// TIA Portal V17 export
// export: Created 2023-12-22T15:02:59.0767996Z, ExportSetting WithDefaults, DisplayName Totally Integrated Automation Portal, DisplayVersion V17, DisplayName TIA Portal Openness, DisplayVersion V17, DisplayName TIA Portal Version Control Interface, DisplayVersion V17, DisplayName STEP 7 Professional, DisplayVersion V17, DisplayName STEP 7 Safety, DisplayVersion V17, DisplayName WinCC Advanced, DisplayVersion V17
FUNCTION_BLOCK "Put_Get"   // FB2, LAD
TITLE = ADDR - удаленный PLC
{ S7_Optimized_Access := 'TRUE' }
VERSION : 0.1
// RD - блок в этом PLC
// stored: AutoNumber true, IsIECCheckEnabled false, IsRetainMemResEnabled false, MemoryReserve 100, SetENOAutomatically false, UDAEnableTagReadback false
   VAR
      GET_SKV_1 { S7_SetPoint := 'True'} : GET;
      GET_SKV_2 { S7_SetPoint := 'True'} : GET;
      GET_SKV_3 { S7_SetPoint := 'True'} : GET;
      GET_SKV_12 { S7_SetPoint := 'True'} : GET;
      GET_SKV_13 { S7_SetPoint := 'True'} : GET;
      GET_SKV_14 { S7_SetPoint := 'True'} : GET;
      GET_SKV_15 { S7_SetPoint := 'True'} : GET;
      GET_SKV_20 { S7_SetPoint := 'True'} : GET;
      GET_SKV_21 { S7_SetPoint := 'True'} : GET;
      GET_SKV_22 { S7_SetPoint := 'True'} : GET;
      GET_SKV_23 { S7_SetPoint := 'True'} : GET;
      PUT_SKV_1 { S7_SetPoint := 'True'} : PUT;
      PUT_SKV_2 { S7_SetPoint := 'True'} : PUT;
      PUT_SKV_3 { S7_SetPoint := 'True'} : PUT;
      PUT_SKV_12 { S7_SetPoint := 'True'} : PUT;
      PUT_SKV_13 { S7_SetPoint := 'True'} : PUT;
      PUT_SKV_14 { S7_SetPoint := 'True'} : PUT;
      PUT_SKV_15 { S7_SetPoint := 'True'} : PUT;
      PUT_SKV_20 { S7_SetPoint := 'True'} : PUT;
      PUT_SKV_21 { S7_SetPoint := 'True'} : PUT;
      PUT_SKV_22 { S7_SetPoint := 'True'} : PUT;
      PUT_SKV_23 { S7_SetPoint := 'True'} : PUT;
      GET_SKD2 { S7_SetPoint := 'True'} : GET;
      PUT_SKD2 { S7_SetPoint := 'True'} : PUT;
   END_VAR
   VAR_TEMP   // added for the SCL form of the ladder/FBD networks
      _w1 : Bool;
      _w2 : Bool;
   END_VAR
BEGIN

REGION Network 1: SKV 1
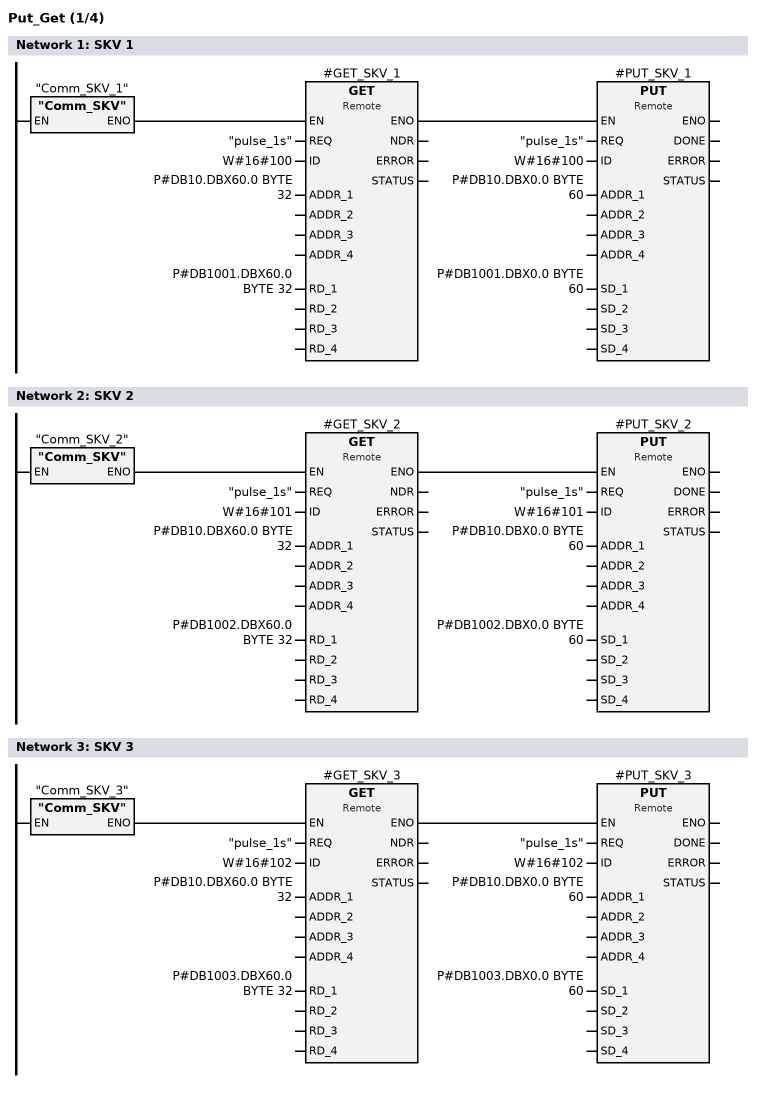
   RUNG wire#powerrail
      "Comm_SKV_1"()
      { S7_Templates := "[remote_type := Remote, local_type := Variant]" } #GET_SKV_1.GET(REQ := "pulse_1s", ID := W#16#100, ADDR_1 := P#DB10.DBX60.0 BYTE 32, ADDR_2 :=, ADDR_3 :=, ADDR_4 :=, RD_1 := P#DB1001.DBX60.0 BYTE 32, RD_2 :=, RD_3 :=, RD_4 :=, NDR =>, ERROR =>, STATUS =>)
      { S7_Templates := "[remote_type := Remote, local_type := Variant]" } #PUT_SKV_1.PUT(REQ := "pulse_1s", ID := W#16#100, ADDR_1 := P#DB10.DBX0.0 BYTE 60, ADDR_2 :=, ADDR_3 :=, ADDR_4 :=, SD_1 := P#DB1001.DBX0.0 BYTE 60, SD_2 :=, SD_3 :=, SD_4 :=, DONE =>, ERROR =>, STATUS =>)
   END_RUNG
   // the same network as SCL:
   "Comm_SKV_1"(ENO => #_w1);   // "Comm_SKV"
   #GET_SKV_1(EN := #_w1,   // GET
              REQ := "pulse_1s",
              ID := W#16#100,
              ADDR_1 := P#DB10.DBX60.0 BYTE 32,
              RD_1 := P#DB1001.DBX60.0 BYTE 32,
              ENO => #_w2);
   IF #_w2 THEN
       #PUT_SKV_1(REQ := "pulse_1s",   // PUT
                  ID := W#16#100,
                  ADDR_1 := P#DB10.DBX0.0 BYTE 60,
                  SD_1 := P#DB1001.DBX0.0 BYTE 60);
   END_IF;
END_REGION

REGION Network 2: SKV 2
   RUNG wire#powerrail
      "Comm_SKV_2"()
      { S7_Templates := "[remote_type := Remote, local_type := Variant]" } #GET_SKV_2.GET(REQ := "pulse_1s", ID := W#16#101, ADDR_1 := P#DB10.DBX60.0 BYTE 32, ADDR_2 :=, ADDR_3 :=, ADDR_4 :=, RD_1 := P#DB1002.DBX60.0 BYTE 32, RD_2 :=, RD_3 :=, RD_4 :=, NDR =>, ERROR =>, STATUS =>)
      { S7_Templates := "[remote_type := Remote, local_type := Variant]" } #PUT_SKV_2.PUT(REQ := "pulse_1s", ID := W#16#101, ADDR_1 := P#DB10.DBX0.0 BYTE 60, ADDR_2 :=, ADDR_3 :=, ADDR_4 :=, SD_1 := P#DB1002.DBX0.0 BYTE 60, SD_2 :=, SD_3 :=, SD_4 :=, DONE =>, ERROR =>, STATUS =>)
   END_RUNG
   // the same network as SCL:
   "Comm_SKV_2"(ENO => #_w1);   // "Comm_SKV"
   #GET_SKV_2(EN := #_w1,   // GET
              REQ := "pulse_1s",
              ID := W#16#101,
              ADDR_1 := P#DB10.DBX60.0 BYTE 32,
              RD_1 := P#DB1002.DBX60.0 BYTE 32,
              ENO => #_w2);
   IF #_w2 THEN
       #PUT_SKV_2(REQ := "pulse_1s",   // PUT
                  ID := W#16#101,
                  ADDR_1 := P#DB10.DBX0.0 BYTE 60,
                  SD_1 := P#DB1002.DBX0.0 BYTE 60);
   END_IF;
END_REGION

REGION Network 3: SKV 3
   RUNG wire#powerrail
      "Comm_SKV_3"()
      { S7_Templates := "[remote_type := Remote, local_type := Variant]" } #GET_SKV_3.GET(REQ := "pulse_1s", ID := W#16#102, ADDR_1 := P#DB10.DBX60.0 BYTE 32, ADDR_2 :=, ADDR_3 :=, ADDR_4 :=, RD_1 := P#DB1003.DBX60.0 BYTE 32, RD_2 :=, RD_3 :=, RD_4 :=, NDR =>, ERROR =>, STATUS =>)
      { S7_Templates := "[remote_type := Remote, local_type := Variant]" } #PUT_SKV_3.PUT(REQ := "pulse_1s", ID := W#16#102, ADDR_1 := P#DB10.DBX0.0 BYTE 60, ADDR_2 :=, ADDR_3 :=, ADDR_4 :=, SD_1 := P#DB1003.DBX0.0 BYTE 60, SD_2 :=, SD_3 :=, SD_4 :=, DONE =>, ERROR =>, STATUS =>)
   END_RUNG
   // the same network as SCL:
   "Comm_SKV_3"(ENO => #_w1);   // "Comm_SKV"
   #GET_SKV_3(EN := #_w1,   // GET
              REQ := "pulse_1s",
              ID := W#16#102,
              ADDR_1 := P#DB10.DBX60.0 BYTE 32,
              RD_1 := P#DB1003.DBX60.0 BYTE 32,
              ENO => #_w2);
   IF #_w2 THEN
       #PUT_SKV_3(REQ := "pulse_1s",   // PUT
                  ID := W#16#102,
                  ADDR_1 := P#DB10.DBX0.0 BYTE 60,
                  SD_1 := P#DB1003.DBX0.0 BYTE 60);
   END_IF;
END_REGION

REGION Network 4: SKV 4
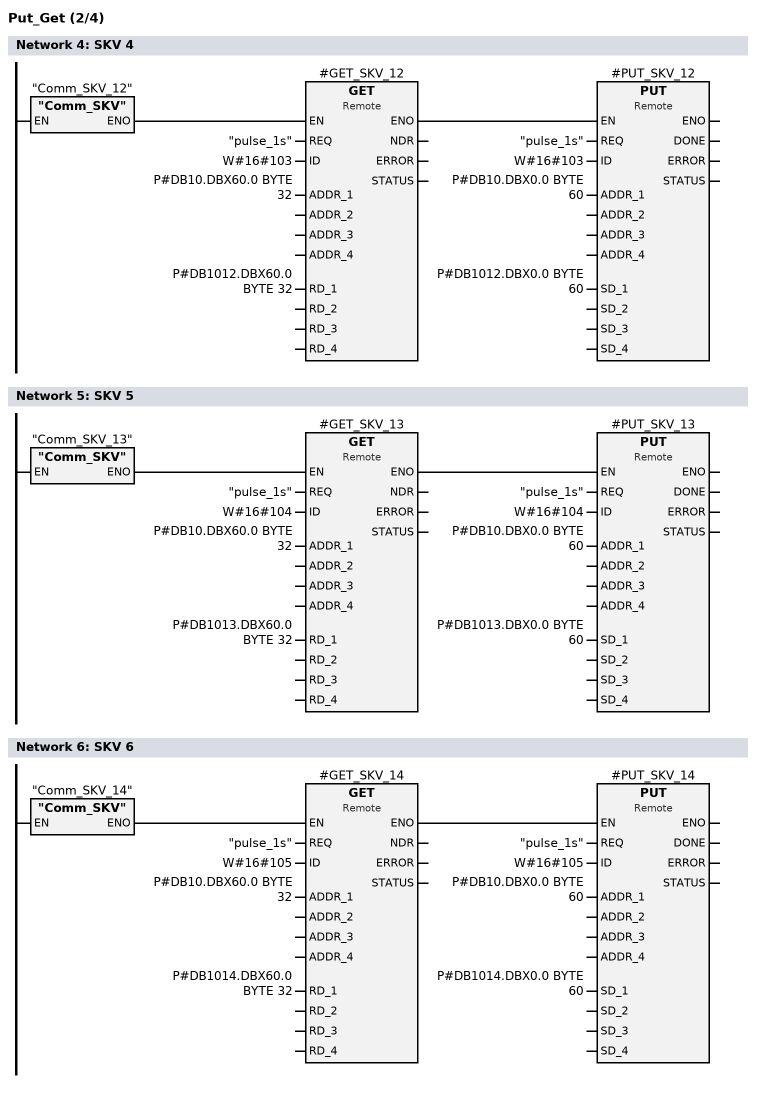
   RUNG wire#powerrail
      "Comm_SKV_12"()
      { S7_Templates := "[remote_type := Remote, local_type := Variant]" } #GET_SKV_12.GET(REQ := "pulse_1s", ID := W#16#103, ADDR_1 := P#DB10.DBX60.0 BYTE 32, ADDR_2 :=, ADDR_3 :=, ADDR_4 :=, RD_1 := P#DB1012.DBX60.0 BYTE 32, RD_2 :=, RD_3 :=, RD_4 :=, NDR =>, ERROR =>, STATUS =>)
      { S7_Templates := "[remote_type := Remote, local_type := Variant]" } #PUT_SKV_12.PUT(REQ := "pulse_1s", ID := W#16#103, ADDR_1 := P#DB10.DBX0.0 BYTE 60, ADDR_2 :=, ADDR_3 :=, ADDR_4 :=, SD_1 := P#DB1012.DBX0.0 BYTE 60, SD_2 :=, SD_3 :=, SD_4 :=, DONE =>, ERROR =>, STATUS =>)
   END_RUNG
   // the same network as SCL:
   "Comm_SKV_12"(ENO => #_w1);   // "Comm_SKV"
   #GET_SKV_12(EN := #_w1,   // GET
               REQ := "pulse_1s",
               ID := W#16#103,
               ADDR_1 := P#DB10.DBX60.0 BYTE 32,
               RD_1 := P#DB1012.DBX60.0 BYTE 32,
               ENO => #_w2);
   IF #_w2 THEN
       #PUT_SKV_12(REQ := "pulse_1s",   // PUT
                   ID := W#16#103,
                   ADDR_1 := P#DB10.DBX0.0 BYTE 60,
                   SD_1 := P#DB1012.DBX0.0 BYTE 60);
   END_IF;
END_REGION

REGION Network 5: SKV 5
   RUNG wire#powerrail
      "Comm_SKV_13"()
      { S7_Templates := "[remote_type := Remote, local_type := Variant]" } #GET_SKV_13.GET(REQ := "pulse_1s", ID := W#16#104, ADDR_1 := P#DB10.DBX60.0 BYTE 32, ADDR_2 :=, ADDR_3 :=, ADDR_4 :=, RD_1 := P#DB1013.DBX60.0 BYTE 32, RD_2 :=, RD_3 :=, RD_4 :=, NDR =>, ERROR =>, STATUS =>)
      { S7_Templates := "[remote_type := Remote, local_type := Variant]" } #PUT_SKV_13.PUT(REQ := "pulse_1s", ID := W#16#104, ADDR_1 := P#DB10.DBX0.0 BYTE 60, ADDR_2 :=, ADDR_3 :=, ADDR_4 :=, SD_1 := P#DB1013.DBX0.0 BYTE 60, SD_2 :=, SD_3 :=, SD_4 :=, DONE =>, ERROR =>, STATUS =>)
   END_RUNG
   // the same network as SCL:
   "Comm_SKV_13"(ENO => #_w1);   // "Comm_SKV"
   #GET_SKV_13(EN := #_w1,   // GET
               REQ := "pulse_1s",
               ID := W#16#104,
               ADDR_1 := P#DB10.DBX60.0 BYTE 32,
               RD_1 := P#DB1013.DBX60.0 BYTE 32,
               ENO => #_w2);
   IF #_w2 THEN
       #PUT_SKV_13(REQ := "pulse_1s",   // PUT
                   ID := W#16#104,
                   ADDR_1 := P#DB10.DBX0.0 BYTE 60,
                   SD_1 := P#DB1013.DBX0.0 BYTE 60);
   END_IF;
END_REGION

REGION Network 6: SKV 6
   RUNG wire#powerrail
      "Comm_SKV_14"()
      { S7_Templates := "[remote_type := Remote, local_type := Variant]" } #GET_SKV_14.GET(REQ := "pulse_1s", ID := W#16#105, ADDR_1 := P#DB10.DBX60.0 BYTE 32, ADDR_2 :=, ADDR_3 :=, ADDR_4 :=, RD_1 := P#DB1014.DBX60.0 BYTE 32, RD_2 :=, RD_3 :=, RD_4 :=, NDR =>, ERROR =>, STATUS =>)
      { S7_Templates := "[remote_type := Remote, local_type := Variant]" } #PUT_SKV_14.PUT(REQ := "pulse_1s", ID := W#16#105, ADDR_1 := P#DB10.DBX0.0 BYTE 60, ADDR_2 :=, ADDR_3 :=, ADDR_4 :=, SD_1 := P#DB1014.DBX0.0 BYTE 60, SD_2 :=, SD_3 :=, SD_4 :=, DONE =>, ERROR =>, STATUS =>)
   END_RUNG
   // the same network as SCL:
   "Comm_SKV_14"(ENO => #_w1);   // "Comm_SKV"
   #GET_SKV_14(EN := #_w1,   // GET
               REQ := "pulse_1s",
               ID := W#16#105,
               ADDR_1 := P#DB10.DBX60.0 BYTE 32,
               RD_1 := P#DB1014.DBX60.0 BYTE 32,
               ENO => #_w2);
   IF #_w2 THEN
       #PUT_SKV_14(REQ := "pulse_1s",   // PUT
                   ID := W#16#105,
                   ADDR_1 := P#DB10.DBX0.0 BYTE 60,
                   SD_1 := P#DB1014.DBX0.0 BYTE 60);
   END_IF;
END_REGION

REGION Network 7: SKV 7
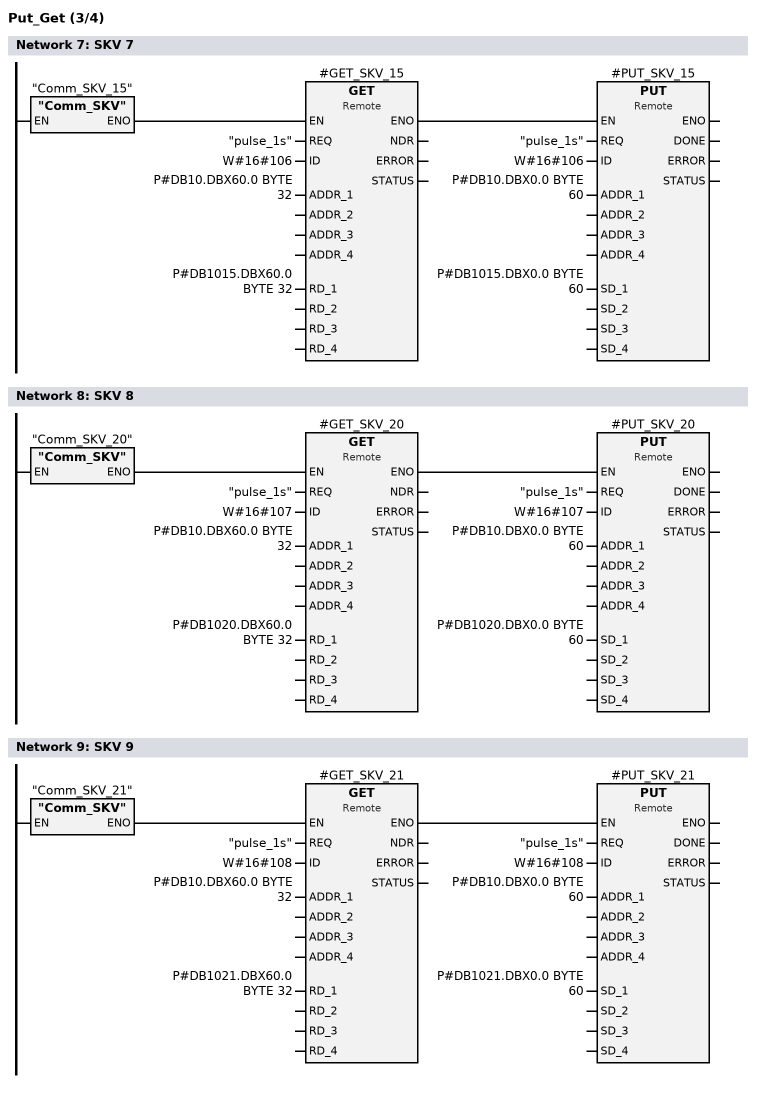
   RUNG wire#powerrail
      "Comm_SKV_15"()
      { S7_Templates := "[remote_type := Remote, local_type := Variant]" } #GET_SKV_15.GET(REQ := "pulse_1s", ID := W#16#106, ADDR_1 := P#DB10.DBX60.0 BYTE 32, ADDR_2 :=, ADDR_3 :=, ADDR_4 :=, RD_1 := P#DB1015.DBX60.0 BYTE 32, RD_2 :=, RD_3 :=, RD_4 :=, NDR =>, ERROR =>, STATUS =>)
      { S7_Templates := "[remote_type := Remote, local_type := Variant]" } #PUT_SKV_15.PUT(REQ := "pulse_1s", ID := W#16#106, ADDR_1 := P#DB10.DBX0.0 BYTE 60, ADDR_2 :=, ADDR_3 :=, ADDR_4 :=, SD_1 := P#DB1015.DBX0.0 BYTE 60, SD_2 :=, SD_3 :=, SD_4 :=, DONE =>, ERROR =>, STATUS =>)
   END_RUNG
   // the same network as SCL:
   "Comm_SKV_15"(ENO => #_w1);   // "Comm_SKV"
   #GET_SKV_15(EN := #_w1,   // GET
               REQ := "pulse_1s",
               ID := W#16#106,
               ADDR_1 := P#DB10.DBX60.0 BYTE 32,
               RD_1 := P#DB1015.DBX60.0 BYTE 32,
               ENO => #_w2);
   IF #_w2 THEN
       #PUT_SKV_15(REQ := "pulse_1s",   // PUT
                   ID := W#16#106,
                   ADDR_1 := P#DB10.DBX0.0 BYTE 60,
                   SD_1 := P#DB1015.DBX0.0 BYTE 60);
   END_IF;
END_REGION

REGION Network 8: SKV 8
   RUNG wire#powerrail
      "Comm_SKV_20"()
      { S7_Templates := "[remote_type := Remote, local_type := Variant]" } #GET_SKV_20.GET(REQ := "pulse_1s", ID := W#16#107, ADDR_1 := P#DB10.DBX60.0 BYTE 32, ADDR_2 :=, ADDR_3 :=, ADDR_4 :=, RD_1 := P#DB1020.DBX60.0 BYTE 32, RD_2 :=, RD_3 :=, RD_4 :=, NDR =>, ERROR =>, STATUS =>)
      { S7_Templates := "[remote_type := Remote, local_type := Variant]" } #PUT_SKV_20.PUT(REQ := "pulse_1s", ID := W#16#107, ADDR_1 := P#DB10.DBX0.0 BYTE 60, ADDR_2 :=, ADDR_3 :=, ADDR_4 :=, SD_1 := P#DB1020.DBX0.0 BYTE 60, SD_2 :=, SD_3 :=, SD_4 :=, DONE =>, ERROR =>, STATUS =>)
   END_RUNG
   // the same network as SCL:
   "Comm_SKV_20"(ENO => #_w1);   // "Comm_SKV"
   #GET_SKV_20(EN := #_w1,   // GET
               REQ := "pulse_1s",
               ID := W#16#107,
               ADDR_1 := P#DB10.DBX60.0 BYTE 32,
               RD_1 := P#DB1020.DBX60.0 BYTE 32,
               ENO => #_w2);
   IF #_w2 THEN
       #PUT_SKV_20(REQ := "pulse_1s",   // PUT
                   ID := W#16#107,
                   ADDR_1 := P#DB10.DBX0.0 BYTE 60,
                   SD_1 := P#DB1020.DBX0.0 BYTE 60);
   END_IF;
END_REGION

REGION Network 9: SKV 9
   RUNG wire#powerrail
      "Comm_SKV_21"()
      { S7_Templates := "[remote_type := Remote, local_type := Variant]" } #GET_SKV_21.GET(REQ := "pulse_1s", ID := W#16#108, ADDR_1 := P#DB10.DBX60.0 BYTE 32, ADDR_2 :=, ADDR_3 :=, ADDR_4 :=, RD_1 := P#DB1021.DBX60.0 BYTE 32, RD_2 :=, RD_3 :=, RD_4 :=, NDR =>, ERROR =>, STATUS =>)
      { S7_Templates := "[remote_type := Remote, local_type := Variant]" } #PUT_SKV_21.PUT(REQ := "pulse_1s", ID := W#16#108, ADDR_1 := P#DB10.DBX0.0 BYTE 60, ADDR_2 :=, ADDR_3 :=, ADDR_4 :=, SD_1 := P#DB1021.DBX0.0 BYTE 60, SD_2 :=, SD_3 :=, SD_4 :=, DONE =>, ERROR =>, STATUS =>)
   END_RUNG
   // the same network as SCL:
   "Comm_SKV_21"(ENO => #_w1);   // "Comm_SKV"
   #GET_SKV_21(EN := #_w1,   // GET
               REQ := "pulse_1s",
               ID := W#16#108,
               ADDR_1 := P#DB10.DBX60.0 BYTE 32,
               RD_1 := P#DB1021.DBX60.0 BYTE 32,
               ENO => #_w2);
   IF #_w2 THEN
       #PUT_SKV_21(REQ := "pulse_1s",   // PUT
                   ID := W#16#108,
                   ADDR_1 := P#DB10.DBX0.0 BYTE 60,
                   SD_1 := P#DB1021.DBX0.0 BYTE 60);
   END_IF;
END_REGION

REGION Network 10: SKV 10
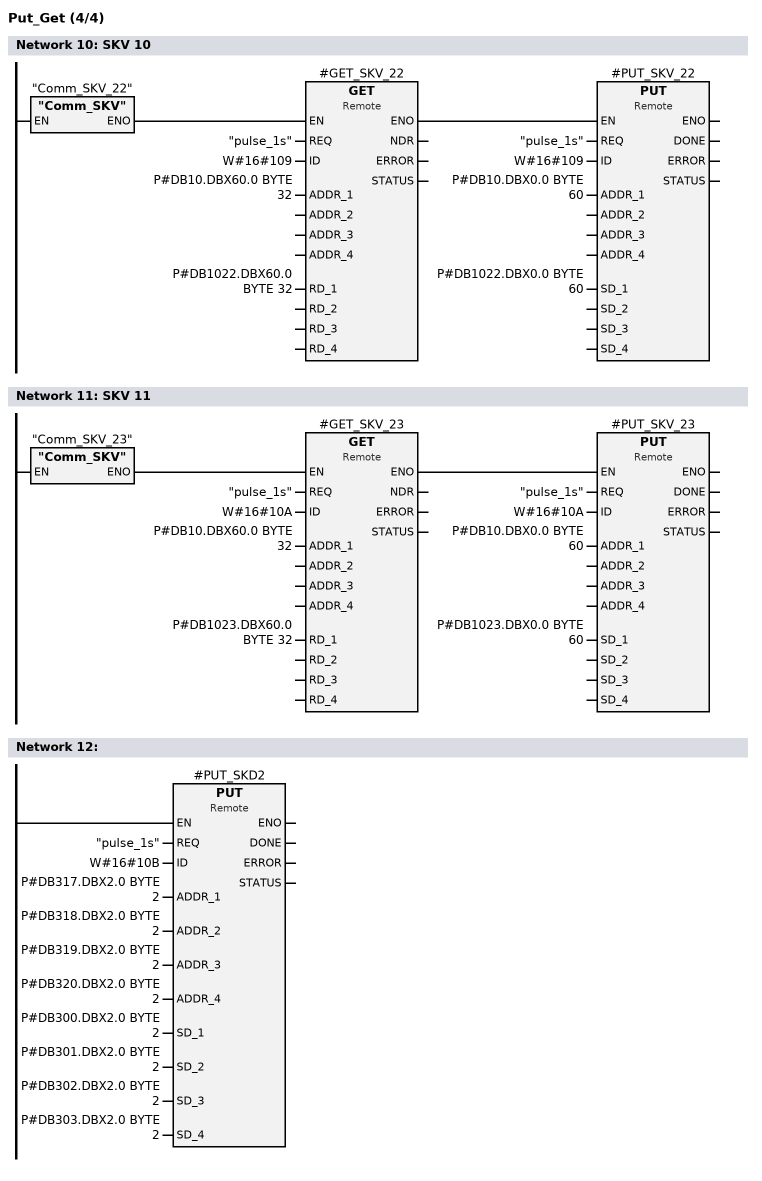
   RUNG wire#powerrail
      "Comm_SKV_22"()
      { S7_Templates := "[remote_type := Remote, local_type := Variant]" } #GET_SKV_22.GET(REQ := "pulse_1s", ID := W#16#109, ADDR_1 := P#DB10.DBX60.0 BYTE 32, ADDR_2 :=, ADDR_3 :=, ADDR_4 :=, RD_1 := P#DB1022.DBX60.0 BYTE 32, RD_2 :=, RD_3 :=, RD_4 :=, NDR =>, ERROR =>, STATUS =>)
      { S7_Templates := "[remote_type := Remote, local_type := Variant]" } #PUT_SKV_22.PUT(REQ := "pulse_1s", ID := W#16#109, ADDR_1 := P#DB10.DBX0.0 BYTE 60, ADDR_2 :=, ADDR_3 :=, ADDR_4 :=, SD_1 := P#DB1022.DBX0.0 BYTE 60, SD_2 :=, SD_3 :=, SD_4 :=, DONE =>, ERROR =>, STATUS =>)
   END_RUNG
   // the same network as SCL:
   "Comm_SKV_22"(ENO => #_w1);   // "Comm_SKV"
   #GET_SKV_22(EN := #_w1,   // GET
               REQ := "pulse_1s",
               ID := W#16#109,
               ADDR_1 := P#DB10.DBX60.0 BYTE 32,
               RD_1 := P#DB1022.DBX60.0 BYTE 32,
               ENO => #_w2);
   IF #_w2 THEN
       #PUT_SKV_22(REQ := "pulse_1s",   // PUT
                   ID := W#16#109,
                   ADDR_1 := P#DB10.DBX0.0 BYTE 60,
                   SD_1 := P#DB1022.DBX0.0 BYTE 60);
   END_IF;
END_REGION

REGION Network 11: SKV 11
   RUNG wire#powerrail
      "Comm_SKV_23"()
      { S7_Templates := "[remote_type := Remote, local_type := Variant]" } #GET_SKV_23.GET(REQ := "pulse_1s", ID := W#16#10A, ADDR_1 := P#DB10.DBX60.0 BYTE 32, ADDR_2 :=, ADDR_3 :=, ADDR_4 :=, RD_1 := P#DB1023.DBX60.0 BYTE 32, RD_2 :=, RD_3 :=, RD_4 :=, NDR =>, ERROR =>, STATUS =>)
      { S7_Templates := "[remote_type := Remote, local_type := Variant]" } #PUT_SKV_23.PUT(REQ := "pulse_1s", ID := W#16#10A, ADDR_1 := P#DB10.DBX0.0 BYTE 60, ADDR_2 :=, ADDR_3 :=, ADDR_4 :=, SD_1 := P#DB1023.DBX0.0 BYTE 60, SD_2 :=, SD_3 :=, SD_4 :=, DONE =>, ERROR =>, STATUS =>)
   END_RUNG
   // the same network as SCL:
   "Comm_SKV_23"(ENO => #_w1);   // "Comm_SKV"
   #GET_SKV_23(EN := #_w1,   // GET
               REQ := "pulse_1s",
               ID := W#16#10A,
               ADDR_1 := P#DB10.DBX60.0 BYTE 32,
               RD_1 := P#DB1023.DBX60.0 BYTE 32,
               ENO => #_w2);
   IF #_w2 THEN
       #PUT_SKV_23(REQ := "pulse_1s",   // PUT
                   ID := W#16#10A,
                   ADDR_1 := P#DB10.DBX0.0 BYTE 60,
                   SD_1 := P#DB1023.DBX0.0 BYTE 60);
   END_IF;
END_REGION

REGION Network 12
   RUNG wire#powerrail
      { S7_Templates := "[remote_type := Remote, local_type := Variant]" } #PUT_SKD2.PUT(REQ := "pulse_1s", ID := W#16#10B, ADDR_1 := P#DB317.DBX2.0 BYTE 2, ADDR_2 := P#DB318.DBX2.0 BYTE 2, ADDR_3 := P#DB319.DBX2.0 BYTE 2, ADDR_4 := P#DB320.DBX2.0 BYTE 2, SD_1 := P#DB300.DBX2.0 BYTE 2, SD_2 := P#DB301.DBX2.0 BYTE 2, SD_3 := P#DB302.DBX2.0 BYTE 2, SD_4 := P#DB303.DBX2.0 BYTE 2, DONE =>, ERROR =>, STATUS =>)
   END_RUNG
   // the same network as SCL:
   #PUT_SKD2(REQ := "pulse_1s",   // PUT
             ID := W#16#10B,
             ADDR_1 := P#DB317.DBX2.0 BYTE 2,
             ADDR_2 := P#DB318.DBX2.0 BYTE 2,
             ADDR_3 := P#DB319.DBX2.0 BYTE 2,
             ADDR_4 := P#DB320.DBX2.0 BYTE 2,
             SD_1 := P#DB300.DBX2.0 BYTE 2,
             SD_2 := P#DB301.DBX2.0 BYTE 2,
             SD_3 := P#DB302.DBX2.0 BYTE 2,
             SD_4 := P#DB303.DBX2.0 BYTE 2);
END_REGION
END_FUNCTION_BLOCK
